FUNCTION_BLOCK EM_Utilities EXTENDS EM_Base IMPLEMENTS I_EM_Utilities
VAR_INPUT
END_VAR
VAR_OUTPUT
END_VAR
VAR
	//Control modules
	s_cmSafetyOk : FB_DigInput;
	s_cm24VdcOk : FB_DigInput;
	s_cmAirPressureOk : FB_DigInput;

	{warning '#TODO: Is it realy necessary to use FB_DigOutput for this, why not using Q'}
	s_cmBeaconLedGreen : FB_DigOutput;
	s_cmBeaconLedYellow : FB_DigOutput;
	s_cmBeaconLedRed : FB_DigOutput;
	//?? see outputs below
	Q_bStaBeaconLedGreen AT %Q* : BOOL;
	Q_bStaBeaconLedYellow AT %Q* : BOOL;
	Q_bStaBeaconLedRed AT %Q* : BOOL;
	
	//States
	s_bStaSafetyOK : BOOL := FALSE;
	s_bSts24VdcOk : BOOL := FALSE;
	s_bStaAirPressureOk : BOOL := FALSE;
	
	s_bStaBeaconRunning : BOOL := FALSE; //green
	s_bStaBeaconWarning : BOOL := FALSE; //yellow
	s_bStaBeaconError : BOOL := FALSE; //red
	
	
	//Hmi
	s_fbHmiLedSafetyOk : FB_HmiLed;
	s_fbHmiLed24VdcOk : FB_HmiLed;
	s_fbHmiLedAirPressureOk : FB_HmiLed;
	s_fbHmiLedBeaconGreen : FB_HmiLed;
	s_fbHmiLedBeaconYellow : FB_HmiLed;
	s_fbHmiLedBeaconRed : FB_HmiLed;
END_VAR

METHOD PROTECTED _m_Alarms : BOOL

IF NOT SUPER^._m_Alarms() THEN
	RETURN;
END_IF
	
_m_Alarms := TRUE;
END_METHOD

METHOD PROTECTED _m_Hmi : BOOL

IF NOT SUPER^._m_Hmi() THEN
	RETURN;
END_IF

//Hmi Leds
s_fbHmiLedSafetyOk(i_bStaLed := s_bStaSafetyOK);
s_fbHmiLed24VdcOk(i_bStaLed := s_bSts24VdcOk);
s_fbHmiLedAirPressureOk(i_bStaLed := s_bStaAirPressureOk);
s_fbHmiLedBeaconGreen(i_bStaLed := s_bStaBeaconRunning);
s_fbHmiLedBeaconYellow(i_bStaLed := s_bStaBeaconWarning);
s_fbHmiLedBeaconRed(i_bStaLed := s_bStaBeaconError);

_m_Hmi := TRUE;
END_METHOD

METHOD PROTECTED _m_Init : BOOL

IF NOT SUPER^._m_Init() THEN
	RETURN;
END_IF

//Control Modules
s_cmSafetyOk.i_stSettings.tmInputDelay := T#1S;
s_cm24VdcOk.i_stSettings.tmInputDelay := T#1S;
s_cmAirPressureOk.i_stSettings.tmInputDelay := T#3S;

s_cmBeaconLedGreen.i_stSettings.bCfgDelay := FALSE;
s_cmBeaconLedGreen.i_stSettings.tmOutputDelay := T#0S;
s_cmBeaconLedYellow.i_stSettings.bCfgDelay := FALSE;
s_cmBeaconLedYellow.i_stSettings.tmOutputDelay := T#0S;
s_cmBeaconLedRed.i_stSettings.bCfgDelay := FALSE;
s_cmBeaconLedRed.i_stSettings.tmOutputDelay := T#0S;

//---------------------------------//	
	
//----------------------------------//	
//Hmi 
s_fbHmiLedSafetyOk.p_bStaVisible := FALSE;
s_fbHmiLedSafetyOk.p_sToHmiDescriptionLed := 'Safety Ok';

s_fbHmiLed24VdcOk.p_bStaVisible := FALSE;
s_fbHmiLed24VdcOk.p_sToHmiDescriptionLed := '24Vdc Ok';

s_fbHmiLedAirPressureOk.p_bStaVisible := FALSE;
s_fbHmiLedAirPressureOk.p_sToHmiDescriptionLed := 'Air pressure Ok';

s_fbHmiLedBeaconGreen.p_bStaVisible := FALSE;
s_fbHmiLedBeaconGreen.p_sToHmiDescriptionLed := 'Beacon green led';

s_fbHmiLedBeaconYellow.p_bStaVisible := FALSE;
s_fbHmiLedBeaconYellow.p_sToHmiDescriptionLed := 'Beacon yellow led';

s_fbHmiLedBeaconRed.p_bStaVisible := FALSE;
s_fbHmiLedBeaconRed.p_sToHmiDescriptionLed := 'Beacon red led';
	
_m_Init := TRUE;
END_METHOD

METHOD PROTECTED _m_Inputs : BOOL

IF NOT SUPER^._m_Inputs() THEN
	RETURN;
END_IF

s_bStaSafetyOK := s_cmSafetyOk.p_bStaInputDelayed;
s_bSts24VdcOk := s_cm24VdcOk.p_bStaInputDelayed;
s_bStaAirPressureOk := s_cmAirPressureOk.p_bStaInputDelayed;

_m_Inputs := TRUE;
END_METHOD

METHOD PROTECTED _m_Modules : BOOL
IF NOT SUPER^._m_Devices() THEN
	RETURN;
END_IF

//Control module
s_cmSafetyOk();
s_cm24VdcOk();
s_cmAirPressureOk();

s_cmBeaconLedGreen.i_bStaOutput := FALSE; //TODO
s_cmBeaconLedYellow.i_bStaOutput := FALSE; //TODO
s_cmBeaconLedRed.i_bStaOutput := 
	NOT(s_bStaSafetyOK) 
	OR NOT(s_bSts24VdcOk)
	OR NOT(s_bStaAirPressureOk);

s_cmBeaconLedGreen();
s_cmBeaconLedYellow();
s_cmBeaconLedRed();
	
_m_Modules := TRUE;
END_METHOD

METHOD PROTECTED _m_Outputs : BOOL

IF NOT SUPER^._m_Outputs() THEN
	RETURN;
END_IF

s_cmBeaconLedGreen.i_bStaOutput := s_bStaBeaconRunning;
s_cmBeaconLedYellow.i_bStaOutput := s_bStaBeaconWarning;
s_cmBeaconLedRed.i_bStaOutput := s_bStaBeaconError;

Q_bStaBeaconLedGreen := s_cmBeaconLedGreen.p_bStaOutput;
Q_bStaBeaconLedYellow := s_cmBeaconLedYellow.p_bStaOutput;
Q_bStaBeaconLedRed := s_cmBeaconLedRed.p_bStaOutput;

_m_Outputs := TRUE;
END_METHOD

PROPERTY PUBLIC p_bStaAirPressureOk : BOOL
GET

p_bStaAirPressureOk := s_bStaAirPressureOk;
END_GET
END_PROPERTY

PROPERTY PUBLIC p_bStaSafetyOK : BOOL
GET

p_bStaSafetyOK := s_bStaSafetyOK;
END_GET
END_PROPERTY

PROPERTY PUBLIC p_bSts24VdcOk : BOOL
GET

p_bSts24VdcOk := s_bSts24VdcOk;
END_GET
END_PROPERTY

END_FUNCTION_BLOCK

(* stored: Version 1.1.0.1, ProductVersion 3.1.4024.12
   POU EM_Utilities: Id {d3bdaf93-23e0-447c-addf-e1fdaa10e5f0}, SpecialFunc None
   Method _m_Alarms: Id {91068a31-fcc6-4281-af61-d7a6e7120f8c}
   Method _m_Hmi: Id {97417a1d-1af2-4f07-b43b-e4325d410b41}
   Method _m_Init: Id {7f1871a0-83c4-4557-ac15-5a15f84be50f}
   Method _m_Inputs: Id {458358e5-23ba-4231-abac-3325a6a209a2}
   Method _m_Modules: Id {97b8a94d-21c8-46ff-ac2c-0f330eabe3be}
   Method _m_Outputs: Id {535a3bcf-7515-4ea2-9150-50d7560b683c}
   Property p_bStaAirPressureOk: Id {0af5c43c-8953-4fa1-af7f-5b3f4e44e13a}
   Get Get: Id {4dede668-7bed-49aa-adc6-f4d7ad59be53}
   Property p_bStaSafetyOK: Id {7ea03187-b7ec-46c2-a694-807e2d1d70bb}
   Get Get: Id {7f5e3440-eaae-47cd-8f92-6961cd1007ef}
   Property p_bSts24VdcOk: Id {4313e908-4780-46b5-aee4-16ddce14fbff}
   Get Get: Id {b2a078c1-b0bd-4ba8-8232-d29d32a14d28} *)
